FUNCTION_BLOCK FB_RangeCheck
VAR_INPUT
	fInput : REAL;
	fLowerLimit : REAL; //lower limit of permission range
	fUpperLimit : REAL; //upper limit of permission range
END_VAR
VAR_OUTPUT
	bPermission : BOOL := TRUE;
END_VAR
VAR
	localDefaultParameters : ST_RangeCheckDefaultParameters;	

	Controller_UpperLimit : FB_CTRL_2POINT;
	Controller_UpperLimit_Parameters : ST_CTRL_2POINT_PARAMS;	
	Controller_LowerLimit : FB_CTRL_2POINT;
	Controller_LowerLimit_Parameters : ST_CTRL_2POINT_PARAMS;	
END_VAR

Controller_UpperLimit_Parameters.fHysteresisRange := localDefaultParameters.fRestoreDifference;
Controller_UpperLimit_Parameters.tCtrlCycleTime := localDefaultParameters.tCtrlCycleTime;
Controller_UpperLimit_Parameters.tTaskCycleTime := localDefaultParameters.tTaskCycleTime;

Controller_UpperLimit(fSetpointValue := fUpperLimit - localDefaultParameters.fRestoreDifference/2,
	fActualValue := fInput,
	eMode := eCTRL_MODE_ACTIVE,
	stParams := Controller_UpperLimit_Parameters);
	
Controller_LowerLimit(fSetpointValue := fInput,
	fActualValue := fLowerLimit + localDefaultParameters.fRestoreDifference/2,
	eMode := eCTRL_MODE_ACTIVE,
	stParams := Controller_UpperLimit_Parameters);
	
bPermission := Controller_UpperLimit.bOut AND Controller_LowerLimit.bOut;

PROPERTY ST_DefaultParameters : REFERENCE TO ST_RangeCheckDefaultParameters
SET
localDefaultParameters := ST_DefaultParameters;
END_SET
END_PROPERTY

END_FUNCTION_BLOCK

(* stored: Version 1.1.0.1, ProductVersion 3.1.4024.10
   POU FB_RangeCheck: Id {5127d44f-afb9-40d0-9273-2d156d799d4a}, SpecialFunc None
   Property ST_DefaultParameters: Id {695e30b8-56ba-4995-b79f-93866d291d34}
   Set Set: Id {04e11d7e-906e-4eac-b62a-a4a5c497dab3} *)
